(* CoDeSys 2.3 export: TEST.EXP *)
(* Libraries: Standard.lib 2.12.10 14:48:34, SYSLIBCALLBACK.LIB 2.12.10 14:48:32 *)

(* PLC configuration (modules and I/O channels)
Hardware configuration [Root] node -1, in %IB0 out %QB0
  K-Bus [K_Bus] node 0, in %IB0 out %QB0
  Fieldbus variables [FB_VARS] node 1, in %IB0 out %QB0
*)

(* POU PLC_PRG, ST *)
PROGRAM PLC_PRG
VAR
	(* BOOL, COIL *)
	COIL1 AT %MX0.0 : BOOL := 0;
	COIL2 AT %MX0.1 : BOOL := 0;
	COIL3 AT %MX0.2 : BOOL := 0;
	COIL4 AT %MX0.3 : BOOL := 0;
	COIL5 AT %MX0.4 : BOOL := 0;
	COIL6 AT %MX0.5 : BOOL := 0;
	COIL7 AT %MX0.6 : BOOL := 0;
	COIL8 AT %MX0.7 : BOOL := 0;

	(* BYTE *)
	BYTE1 AT %MB0 : BYTE := 0;
	BYTE2 AT %MB1 : BYTE := 0;
	BYTE3 AT %MB2 : BYTE := 0;
	BYTE4 AT %MB3 : BYTE := 0;
	BYTE5 AT %MB4 : BYTE := 0;

	(* INT *)
	INT1 AT %MW0 : INT := 0;
	INT2 AT %MW1 : INT := 0;
	INT3 AT %MW2 : INT := 0;
	INT4 AT %MW3 : INT := 0;
	INT5 AT %MW4 : INT := 0;

	(* WORD *)
	WORD1 AT %MW0 : WORD := 0;
	WORD2 AT %MW1 : WORD := 0;
	WORD3 AT %MW2 : WORD := 0;
	WORD4 AT %MW3 : WORD := 0;
	WORD5 AT %MW4 : WORD := 0;

	(* DINT *)
	DINT1 AT %MD0 : DINT := 0;
	DINT2 AT %MD1 : DINT := 0;
	DINT3 AT %MD2 : DINT := 0;
	DINT4 AT %MD3 : DINT := 0;
	DINT5 AT %MD4 : DINT := 0;

	(* DWORD *)
	DWORD1 AT %MD0 : DWORD := 0;
	DWORD2 AT %MD1 : DWORD := 0;
	DWORD3 AT %MD2 : DWORD := 0;
	DWORD4 AT %MD3 : DWORD := 0;
	DWORD5 AT %MD4 : DWORD := 0;

	(* REAL *)
	REAL1 AT %MD0 : REAL := 0;
	REAL2 AT %MD1 : REAL := 0;
	REAL3 AT %MD2 : REAL := 0;
	REAL4 AT %MD3 : REAL := 0;
	REAL5 AT %MD4 : REAL := 0;

	(* String *)
	STRING1 AT %MW0 : STRING := 'Hello word!!!';
END_VAR
(* Something to do *)
;
END_PROGRAM
